// TIA Portal project "Thor_V1" (V15)

(* hardware
DEVICE "S71500/ET200MP station_1"  S7-1500 station
   slot 0: "Rail_0"  Rack  6ES7 590-1***0-0AA0
   slot 1: "PLC_1"  CPU 1516F-3 PN/DP  6ES7 516-3FN01-0AB0  V2.5
      slot 3: "CPU display_1"  6ES7591-1BA00-0AA0
   slot 2: "DI 16x24VDC HF"  DI 16x24VDC HF  6ES7 521-1BH00-0AB0  V2.1
   slot 3: "DQ 16x24VDC/0.5A ST_1"  DQ 16x24VDC/0.5A ST  6ES7 522-1BH00-0AB0  V2.0
DEVICE "GSD device_1"  GSD.Device.PN
   slot 0: "Rack"  Rack  V1.0
   slot 0: "InSight"  In-Sight ISM1XXX  ISM1XXX-XX  4.10.0
      slot 0: "In-Sight ISM1XXX"  In-Sight ISM1XXX  4.10.0
      slot 1: "Interface"  Interface
         slot 1: "Port 1"  Port 1
   slot 1: "Acquisition Control_1"  Acquisition Control  5.1.1
      slot 0: "Acquisition Control"  Acquisition Control  5.1.1
   slot 2: "Acquisition Status_1"  Acquisition Status  5.1.1
      slot 0: "Acquisition Status"  Acquisition Status  5.1.1
   slot 3: "Inspection Control_1"  Inspection Control  5.1.1
      slot 0: "Inspection Control"  Inspection Control  5.1.1
   slot 4: "Inspection Status_1"  Inspection Status  4.10.0
      slot 0: "Inspection Status"  Inspection Status  4.10.0
   slot 5: "Job Control_1"  Job Control  4.10.0
      slot 0: "Job Control"  Job Control  4.10.0
   slot 6: "SoftEvent Control_1"  SoftEvent Control  4.10.0
      slot 0: "SoftEvent Control"  SoftEvent Control  4.10.0
   slot 7: "User Data - 64 bytes_1"  User Data - 64 bytes  5.1.1
      slot 0: "User Data - 64 bytes"  User Data - 64 bytes  5.1.1
   slot 8: "Results - 64 bytes_1"  Results - 64 bytes  5.1.1
      slot 0: "Results - 64 bytes"  Results - 64 bytes  5.1.1
*)

// ===== PLC "PLC_1"  CPU 1516F-3 PN/DP =====

VAR_GLOBAL   // PLC tag table "Default tag table"
   "x" AT %MW10 : Int;
   "y" AT %MW12 : Int;
   "Tag_1" AT %M0.0 : Bool;
   "Tag_2" AT %M0.1 : Bool;
   "Tag_3" AT %M1.0 : Bool;
   "Tag_4" AT %M1.1 : Bool;
   "Tag_5" AT %M1.2 : Bool;
   "Tag_6" AT %M0.5 : Bool;
   "System_Byte" AT %MB1 : Byte;
   "FirstScan" AT %M1.0 : Bool;
   "DiagStatusUpdate" AT %M1.1 : Bool;
   "AlwaysTRUE" AT %M1.2 : Bool;
   "AlwaysFALSE" AT %M1.3 : Bool;
   "Clock_Byte" AT %MB0 : Byte;
   "Clock_10Hz" AT %M0.0 : Bool;
   "Clock_5Hz" AT %M0.1 : Bool;
   "Clock_2.5Hz" AT %M0.2 : Bool;
   "Clock_2Hz" AT %M0.3 : Bool;
   "Clock_1.25Hz" AT %M0.4 : Bool;
   "Clock_1Hz" AT %M0.5 : Bool;
   "Clock_0.625Hz" AT %M0.6 : Bool;
   "Clock_0.5Hz" AT %M0.7 : Bool;
   "Tag_7" AT %M100.0 : Bool;
   "Tag_8" AT %M100.1 : Bool;
   "Tag_9" AT %M100.2 : Bool;
   "Tag_10" AT %M100.3 : Bool;
   "brak_elementu" AT %M6.0 : Bool;
   "wyslij_dane" AT %M10.0 : Bool;
   "Tag_12" AT %M10.1 : Bool;
   "wysylane_dane" AT %MW200 : Word;
   "wysylane" AT %MW202 : Int;
   "Tag_11" AT %M202.0 : Bool;
   "Tag_13" AT %M120.0 : Bool;
   "Tag_14" AT %M140.5 : Bool;
   "Tag_15" AT %M130.0 : Bool;
   "Tag_16" AT %M2.0 : Bool;
   "Tag_17" AT %M2.1 : Bool;
   "y_w_10" AT %M2.2 : Bool;
   "Tag_18" AT %M2.3 : Bool;
   "M4.0" AT %M2.4 : Bool;
   "x_w_10" AT %M2.5 : Bool;
   "Tag_20" AT %M2.6 : Bool;
   "Tag_21" AT %M2.7 : Bool;
   "y_m_-10" AT %M3.0 : Bool;
   "Tag_22" AT %M3.1 : Bool;
   "Tag_23" AT %M3.2 : Bool;
   "x_m_-10" AT %M3.3 : Bool;
   "Tag_24" AT %M3.4 : Bool;
   "Tag_25" AT %M3.5 : Bool;
   "y_stop" AT %M3.6 : Bool;
   "Tag_26" AT %M3.7 : Bool;
   "x_stop" AT %M4.1 : Bool;
   "y_send" AT %M5.0 : Bool;
   "x_send" AT %M5.1 : Bool;
   "Tag_19" AT %M20.0 : Bool;
   "Tag_27" AT %M57.0 : Bool;
   "Tag_28" AT %M57.5 : Bool;
   "Tag_29" AT %M18.6 : Bool;
   "sensor" AT %I74.0 : Bool;
   "Tag_30" AT %M27.0 : Bool;
   "Tag_31" AT %M27.1 : Bool;
   "silnik" AT %Q68.7 : Bool;
   "silnik(1)" AT %Q68.0 : Bool;
   "Motor" AT %Q68.1 : Bool;
END_VAR

VAR_GLOBAL   // PLC tag table "Kamerka"
   "detection-TriggerEnable" AT %Q0.0 : Bool;
   "detection-Trigger" AT %Q0.1 : Bool;
   "detection-ClearExposureComplete" AT %Q0.2 : Bool;
   "detection-SetOffline" AT %Q0.7 : Bool;
   "detection-TriggerReady" AT %I0.0 : Bool;
   "detection-TriggerAck" AT %I0.1 : Bool;
   "detection-ExposureComplete" AT %I0.2 : Bool;
   "detection-MissedAcq" AT %I0.3 : Bool;
   "detection-OfflineReason(0)" AT %I0.4 : Bool;
   "detection-OfflineReason(1)" AT %I0.5 : Bool;
   "detection-OfflineReason(2)" AT %I0.6 : Bool;
   "detection-Online" AT %I0.7 : Bool;
   "detection-AcquisitionID" AT %IW1 : Int;
   "detection-BufferResultsEnable" AT %Q1.0 : Bool;
   "detection-InspectionResultsAck" AT %Q1.1 : Bool;
   "detection-SetUserData" AT %Q1.2 : Bool;
   "detection-ExecuteCommand/JobLoad" AT %Q1.3 : Bool;
   "detection-ClearError" AT %Q1.7 : Bool;
   "detection-SystemBusy" AT %I3.0 : Bool;
   "detection-InspectionCompleted" AT %I3.1 : Bool;
   "detection-ResultsBufferOverrun" AT %I3.2 : Bool;
   "detection-ResultsValid" AT %I3.3 : Bool;
   "detection-CommandExecuting" AT %I3.4 : Bool;
   "detection-CommandCompleted" AT %I3.5 : Bool;
   "detection-CommandFailed" AT %I3.6 : Bool;
   "detection-SetUserDataAck" AT %I3.7 : Bool;
   "detection-JobPass" AT %I4.0 : Bool;
   "detection-TestRunReady" AT %I4.1 : Bool;
   "detection-Error" AT %I4.7 : Bool;
   "detection-ErrorCode" AT %IW5 : Word;
   "detection-CommandInput" AT %IW5 : Word;
   "detection-CommandOutput" AT %QW2 : Word;
   "detection-SoftEvent[0]" AT %Q3.0 : Bool;
   "detection-SoftEvent[1]" AT %Q3.1 : Bool;
   "detection-SoftEvent[2]" AT %Q3.2 : Bool;
   "detection-SoftEvent[3]" AT %Q3.3 : Bool;
   "detection-SoftEvent[4]" AT %Q3.4 : Bool;
   "detection-SoftEvent[5]" AT %Q3.5 : Bool;
   "detection-SoftEvent[6]" AT %Q3.6 : Bool;
   "detection-SoftEvent[7]" AT %Q3.7 : Bool;
   "detection-SoftEventAck[0]" AT %I2.0 : Bool;
   "detection-SoftEventAck[1]" AT %I2.1 : Bool;
   "detection-SoftEventAck[2]" AT %I2.2 : Bool;
   "detection-SoftEventAck[3]" AT %I2.3 : Bool;
   "detection-SoftEventAck[4]" AT %I2.4 : Bool;
   "detection-SoftEventAck[5]" AT %I2.5 : Bool;
   "detection-SoftEventAck[6]" AT %I2.6 : Bool;
   "detection-SoftEventAck[7]" AT %I2.7 : Bool;
   "detection-UserData[0]" AT %QB4 : Char;
   "detection-UserData[1]" AT %QB5 : Byte;
   "detection-UserData[2]" AT %QB6 : Byte;
   "detection-UserData[3]" AT %QB7 : Byte;
   "detection-UserData[4]" AT %QB8 : Byte;
   "detection-UserData[5]" AT %QB9 : Byte;
   "detection-UserData[6]" AT %QB10 : Byte;
   "detection-UserData[7]" AT %QB11 : Byte;
   "detection-UserData[8]" AT %QB12 : Byte;
   "detection-UserData[9]" AT %QB13 : Byte;
   "detection-UserData[10]" AT %QB14 : Byte;
   "detection-UserData[11]" AT %QB15 : Byte;
   "detection-UserData[12]" AT %QB16 : Byte;
   "detection-UserData[13]" AT %QB17 : Byte;
   "detection-UserData[14]" AT %QB18 : Byte;
   "detection-UserData[15]" AT %QB19 : Byte;
   "detection-InspectionID" AT %IW6 : Word;
   "detection-InspectionResultsCode" AT %IW8 : Int;
   "x_sub" AT %IW10 : Int;
   "y_sub" AT %IW12 : Int;
END_VAR

DATA_BLOCK "Data_block_1"   // DB1
{ S7_Optimized_Access := 'TRUE' }
VERSION : 0.1
   VAR
      data_y : Char := 'Y';
      data_x : Char := 'X';
   END_VAR
BEGIN
END_DATA_BLOCK

// folder: System blocks/Program resources

DATA_BLOCK "IEC_Timer_0_DB"   // DB2
{ S7_Optimized_Access := 'TRUE' }
AUTHOR : Simatic
FAMILY : IEC
NAME : IEC_TMR
VERSION : 1.0
// stored: InstanceOfName IEC_TIMER
"IEC_TIMER"
BEGIN
END_DATA_BLOCK

DATA_BLOCK "PLC_1_Send_DB"   // DB4
{ S7_Optimized_Access := 'TRUE' }
AUTHOR : SIMATIC
FAMILY : MC7Plus
NAME : TC_IP_v4
VERSION : 1.0
// stored: InstanceOfName TCON_IP_v4
"TCON_IP_v4"
BEGIN
   ID := 1;
   InterfaceId := 64;
   RemotePort := 2000;
   ActiveEstablished := true;
   RemoteAddress.ADDR[1] := 192;
   RemoteAddress.ADDR[2] := 168;
   RemoteAddress.ADDR[4] := 30;
END_DATA_BLOCK

// folder: (top level)

ORGANIZATION_BLOCK "Main"   // OB1, LAD, ProgramCycle
TITLE = "Main Program Sweep (Cycle)"
{ S7_Optimized_Access := 'TRUE' }
VERSION : 0.1
   VAR_INPUT
      Initial_Call : Bool;   // Initial call of this OB
      Remanence : Bool;   // =True, if remanent data are available
   END_VAR
   VAR_TEMP   // added for the SCL form of the ladder/FBD networks
      _w1 : Bool;
   END_VAR
BEGIN

REGION Network 1
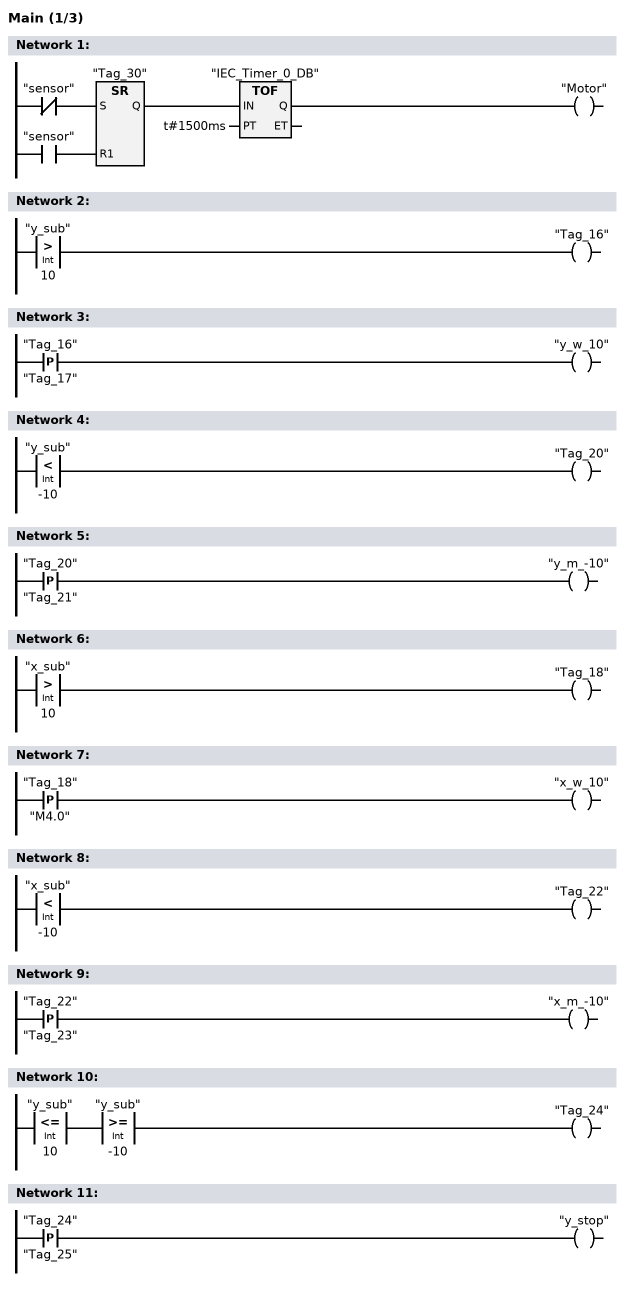
   IF NOT "sensor" THEN
       "Tag_30" := TRUE;   // SR flip-flop
   END_IF;
   IF "sensor" THEN "Tag_30" := FALSE; END_IF;
   "IEC_Timer_0_DB".TOF(IN := "Tag_30", PT := t#1500ms);
   "Motor" := "IEC_Timer_0_DB".Q;
END_REGION

REGION Network 2
   RUNG wire#powerrail
      { S7_Templates := "SrcType := Int" } GT_Contact(in1 := "y_sub", in2 := 10)
      Coil( "Tag_16" )
   END_RUNG
   // the same network as SCL:
   "Tag_16" := "y_sub" > 10;
END_REGION

REGION Network 3
   RUNG wire#powerrail
      P_Contact(operand := "Tag_16", bit := "Tag_17")
      Coil( "y_w_10" )
   END_RUNG
   // the same network as SCL:
   #_w1 := "Tag_16" AND NOT "Tag_17";   // rising edge of "Tag_16"
   "Tag_17" := "Tag_16";
   "y_w_10" := #_w1;
END_REGION

REGION Network 4
   RUNG wire#powerrail
      { S7_Templates := "SrcType := Int" } LT_Contact(in1 := "y_sub", in2 := -10)
      Coil( "Tag_20" )
   END_RUNG
   // the same network as SCL:
   "Tag_20" := "y_sub" < (-10);
END_REGION

REGION Network 5
   RUNG wire#powerrail
      P_Contact(operand := "Tag_20", bit := "Tag_21")
      Coil( "y_m_-10" )
   END_RUNG
   // the same network as SCL:
   #_w1 := "Tag_20" AND NOT "Tag_21";   // rising edge of "Tag_20"
   "Tag_21" := "Tag_20";
   "y_m_-10" := #_w1;
END_REGION

REGION Network 6
   RUNG wire#powerrail
      { S7_Templates := "SrcType := Int" } GT_Contact(in1 := "x_sub", in2 := 10)
      Coil( "Tag_18" )
   END_RUNG
   // the same network as SCL:
   "Tag_18" := "x_sub" > 10;
END_REGION

REGION Network 7
   RUNG wire#powerrail
      P_Contact(operand := "Tag_18", bit := "M4.0")
      Coil( "x_w_10" )
   END_RUNG
   // the same network as SCL:
   #_w1 := "Tag_18" AND NOT "M4.0";   // rising edge of "Tag_18"
   "M4.0" := "Tag_18";
   "x_w_10" := #_w1;
END_REGION

REGION Network 8
   RUNG wire#powerrail
      { S7_Templates := "SrcType := Int" } LT_Contact(in1 := "x_sub", in2 := -10)
      Coil( "Tag_22" )
   END_RUNG
   // the same network as SCL:
   "Tag_22" := "x_sub" < (-10);
END_REGION

REGION Network 9
   RUNG wire#powerrail
      P_Contact(operand := "Tag_22", bit := "Tag_23")
      Coil( "x_m_-10" )
   END_RUNG
   // the same network as SCL:
   #_w1 := "Tag_22" AND NOT "Tag_23";   // rising edge of "Tag_22"
   "Tag_23" := "Tag_22";
   "x_m_-10" := #_w1;
END_REGION

REGION Network 10
   RUNG wire#powerrail
      { S7_Templates := "SrcType := Int" } LE_Contact(in1 := "y_sub", in2 := 10)
      { S7_Templates := "SrcType := Int" } GE_Contact(in1 := "y_sub", in2 := -10)
      Coil( "Tag_24" )
   END_RUNG
   // the same network as SCL:
   "Tag_24" := ("y_sub" <= 10) AND ("y_sub" >= (-10));
END_REGION

REGION Network 11
   RUNG wire#powerrail
      P_Contact(operand := "Tag_24", bit := "Tag_25")
      Coil( "y_stop" )
   END_RUNG
   // the same network as SCL:
   #_w1 := "Tag_24" AND NOT "Tag_25";   // rising edge of "Tag_24"
   "Tag_25" := "Tag_24";
   "y_stop" := #_w1;
END_REGION

REGION Network 12
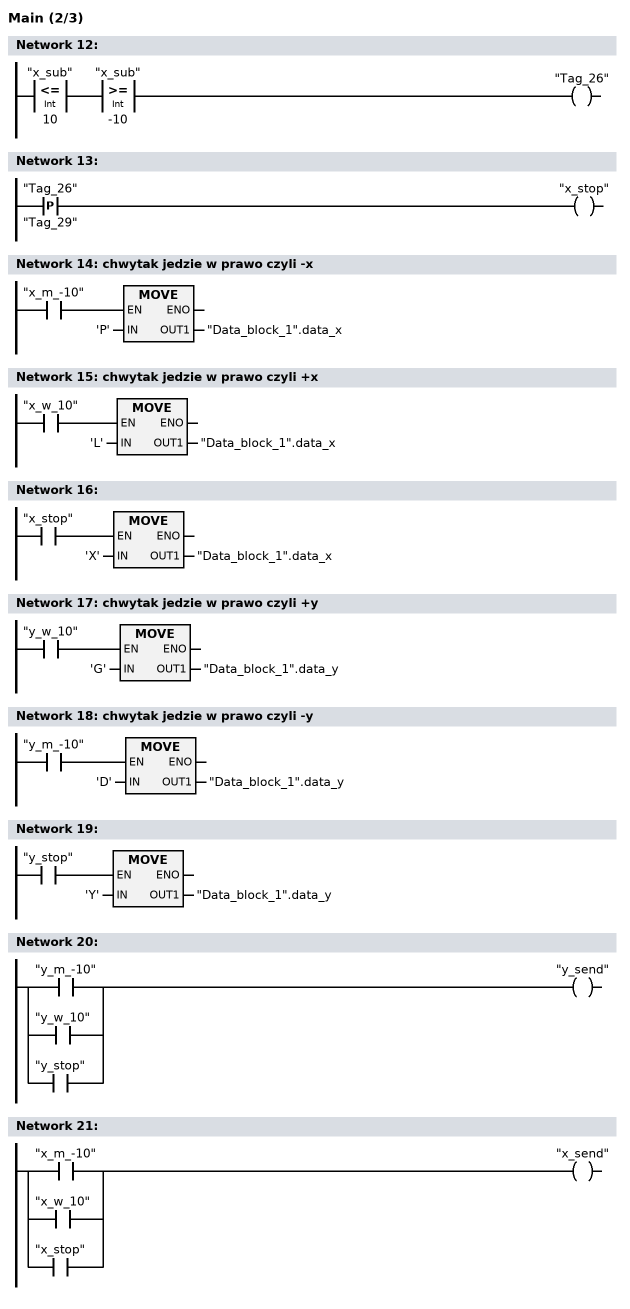
   RUNG wire#powerrail
      { S7_Templates := "SrcType := Int" } LE_Contact(in1 := "x_sub", in2 := 10)
      { S7_Templates := "SrcType := Int" } GE_Contact(in1 := "x_sub", in2 := -10)
      Coil( "Tag_26" )
   END_RUNG
   // the same network as SCL:
   "Tag_26" := ("x_sub" <= 10) AND ("x_sub" >= (-10));
END_REGION

REGION Network 13
   RUNG wire#powerrail
      P_Contact(operand := "Tag_26", bit := "Tag_29")
      Coil( "x_stop" )
   END_RUNG
   // the same network as SCL:
   #_w1 := "Tag_26" AND NOT "Tag_29";   // rising edge of "Tag_26"
   "Tag_29" := "Tag_26";
   "x_stop" := #_w1;
END_REGION

REGION Network 14: chwytak jedzie w prawo czyli -x
   RUNG wire#powerrail
      Contact( "x_m_-10" )
      Move(in := 'P', out1 => "Data_block_1".data_x)
   END_RUNG
   // the same network as SCL:
   IF "x_m_-10" THEN "Data_block_1".data_x := 'P'; END_IF;
END_REGION

REGION Network 15: chwytak jedzie w prawo czyli +x
   RUNG wire#powerrail
      Contact( "x_w_10" )
      Move(in := 'L', out1 => "Data_block_1".data_x)
   END_RUNG
   // the same network as SCL:
   IF "x_w_10" THEN "Data_block_1".data_x := 'L'; END_IF;
END_REGION

REGION Network 16
   RUNG wire#powerrail
      Contact( "x_stop" )
      Move(in := 'X', out1 => "Data_block_1".data_x)
   END_RUNG
   // the same network as SCL:
   IF "x_stop" THEN "Data_block_1".data_x := 'X'; END_IF;
END_REGION

REGION Network 17: chwytak jedzie w prawo czyli +y
   RUNG wire#powerrail
      Contact( "y_w_10" )
      Move(in := 'G', out1 => "Data_block_1".data_y)
   END_RUNG
   // the same network as SCL:
   IF "y_w_10" THEN "Data_block_1".data_y := 'G'; END_IF;
END_REGION

REGION Network 18: chwytak jedzie w prawo czyli -y
   RUNG wire#powerrail
      Contact( "y_m_-10" )
      Move(in := 'D', out1 => "Data_block_1".data_y)
   END_RUNG
   // the same network as SCL:
   IF "y_m_-10" THEN "Data_block_1".data_y := 'D'; END_IF;
END_REGION

REGION Network 19
   RUNG wire#powerrail
      Contact( "y_stop" )
      Move(in := 'Y', out1 => "Data_block_1".data_y)
   END_RUNG
   // the same network as SCL:
   IF "y_stop" THEN "Data_block_1".data_y := 'Y'; END_IF;
END_REGION

REGION Network 20
   RUNG wire#powerrail
      Contact( "y_m_-10" )
      wire#w1
      Coil( "y_send" )
   END_RUNG
   RUNG wire#powerrail
      Contact( "y_w_10" )
   END_RUNG wire#w1
   RUNG wire#powerrail
      Contact( "y_stop" )
   END_RUNG wire#w1
   // the same network as SCL:
   "y_send" := "y_m_-10" OR "y_w_10" OR "y_stop";
END_REGION

REGION Network 21
   RUNG wire#powerrail
      Contact( "x_m_-10" )
      wire#w1
      Coil( "x_send" )
   END_RUNG
   RUNG wire#powerrail
      Contact( "x_w_10" )
   END_RUNG wire#w1
   RUNG wire#powerrail
      Contact( "x_stop" )
   END_RUNG wire#w1
   // the same network as SCL:
   "x_send" := "x_m_-10" OR "x_w_10" OR "x_stop";
END_REGION

REGION Network 22
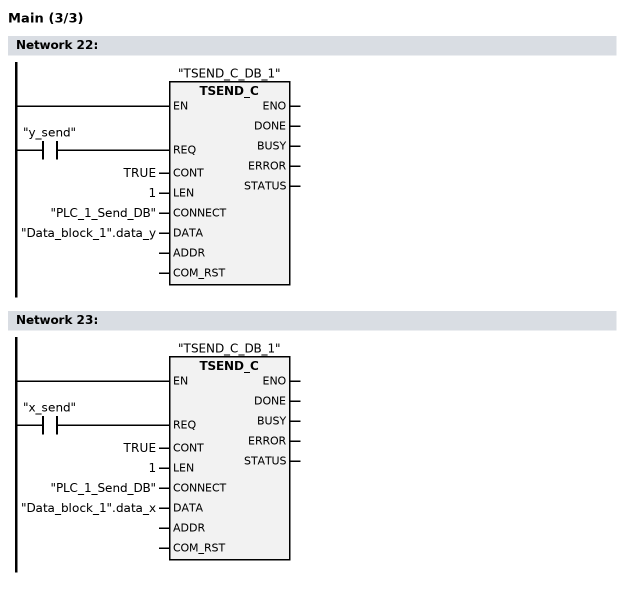
   "TSEND_C_DB_1"(REQ := "y_send",   // TSEND_C
                  CONT := TRUE,
                  LEN := 1,
                  CONNECT := "PLC_1_Send_DB",
                  DATA := "Data_block_1".data_y);
END_REGION

REGION Network 23
   "TSEND_C_DB_1"(REQ := "x_send",   // TSEND_C
                  CONT := TRUE,
                  LEN := 1,
                  CONNECT := "PLC_1_Send_DB",
                  DATA := "Data_block_1".data_x);
END_REGION
END_ORGANIZATION_BLOCK